// TIA Portal V16 export
// export: Created 2023-08-28T09:37:31.5256679Z, ExportSetting WithDefaults, DisplayName Totally Integrated Automation Portal, DisplayVersion V16 Update 6, DisplayName TIA Portal Version Control Interface, DisplayVersion V16 Update 2, DisplayName TIA Portal Openness, DisplayVersion V16 Update 6, DisplayName STEP 7 Professional, DisplayVersion V16 Update 6, DisplayName STEP 7 Safety, DisplayVersion V16, DisplayName WinCC Advanced, DisplayVersion V16 Update 6
FUNCTION_BLOCK "00_S_AutomaticPIDReset"   // FB22, LAD
{ S7_Optimized_Access := 'TRUE' }
VERSION : 0.1
// stored: AutoNumber true, IsIECCheckEnabled false, IsRetainMemResEnabled false, MemoryReserve 250, SetENOAutomatically false, UDAEnableTagReadback false
   VAR_INPUT
      State : Int;
      Error : DWord;
   END_VAR
   VAR_OUTPUT
      LastError : DWord;
      StateBeforeError : Int;
      "sRet.i_Mode" : Int;
   END_VAR
   VAR_TEMP   // added for the SCL form of the ladder/FBD networks
      _w1 : Bool;
   END_VAR
BEGIN

REGION Network 1: State Before Error
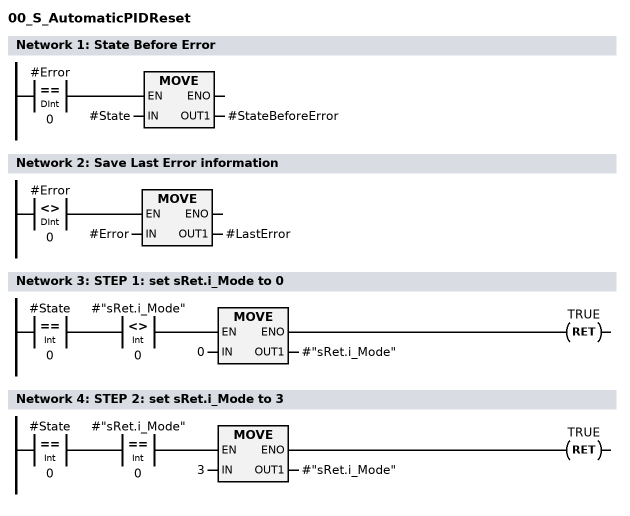
   RUNG wire#powerrail
      { S7_Templates := "SrcType := DInt" } EQ_Contact(in1 := #Error, in2 := 0)
      { S7_GenerateENO := "TRUE" } Move(in := #State, out1 => #StateBeforeError)
   END_RUNG
   // the same network as SCL:
   IF #Error = 0 THEN #StateBeforeError := #State; END_IF;
END_REGION

REGION Network 2: Save Last Error information
   RUNG wire#powerrail
      { S7_Templates := "SrcType := DInt" } NE_Contact(in1 := #Error, in2 := 0)
      { S7_GenerateENO := "TRUE" } Move(in := #Error, out1 => #LastError)
   END_RUNG
   // the same network as SCL:
   IF #Error <> 0 THEN #LastError := #Error; END_IF;
END_REGION

REGION Network 3: STEP 1: set sRet.i_Mode to 0
   // ENO of a box is taken as its EN; it also drops when the box reports an error
   #_w1 := (#State = 0) AND (#"sRet.i_Mode" <> 0);
   IF #_w1 THEN
       #"sRet.i_Mode" := 0;
       ENO := TRUE;
       RETURN;
   END_IF;
END_REGION

REGION Network 4: STEP 2: set sRet.i_Mode to 3
   // ENO of a box is taken as its EN; it also drops when the box reports an error
   #_w1 := (#State = 0) AND (#"sRet.i_Mode" = 0);
   IF #_w1 THEN
       #"sRet.i_Mode" := 3;
       ENO := TRUE;
       RETURN;
   END_IF;
END_REGION
END_FUNCTION_BLOCK
